FUNCTION_BLOCK LiftModel (* Basic Function Block Type *)
  (* Standard: 61499-2 *)
  (* Version 0.0, 4/20/2019, vshatrov, nxtControl GmbH, Template *)
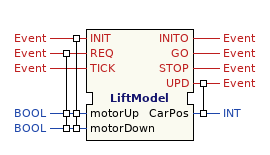
  EVENT_INPUT
    INIT WITH motorUp, motorDown; (* Initialization Request *)
    REQ WITH motorUp, motorDown; (* Normal Execution Request *)
    TICK;
  END_EVENT
  EVENT_OUTPUT
    INITO;
    GO; (* Initialization Confirm *)
    STOP; (* Execution Confirmation *)
    UPD WITH CarPos;
  END_EVENT
  VAR_INPUT
    motorUp : BOOL; (* Input event qualifier *)
    motorDown : BOOL;
  END_VAR
  VAR_OUTPUT
    CarPos : INT; (* Output event qualifier *)
  END_VAR
  VAR
    Position : DINT;
    direction : DINT;
  END_VAR
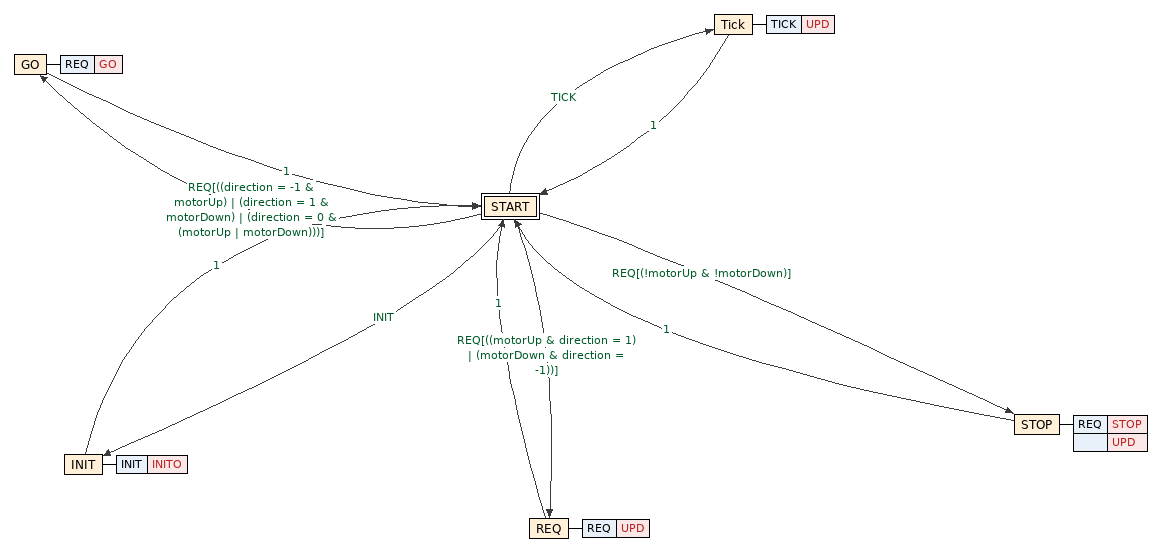
  EC_STATES
    START; (* Initial State *)
    INIT : INIT -> INITO; (* Initialization *)
    REQ : REQ -> UPD; (* Normal execution *)
    Tick : TICK -> UPD;
    GO : REQ -> GO;
    STOP : REQ -> STOP, -> UPD;
  END_STATES
  EC_TRANSITIONS
    START TO INIT := INIT;
    INIT TO START := 1;
    START TO GO := REQ[((direction = -1 & motorUp) | (direction = 1 & motorDown) | (direction = 0 & (motorUp | motorDown)))];
    START TO Tick := TICK;
    Tick TO START := 1;
    START TO STOP := REQ[(!motorUp & !motorDown)];
    GO TO START := 1;
    STOP TO START := 1;
    START TO REQ := REQ[((motorUp & direction = 1) | (motorDown & direction = -1))];
    REQ TO START := 1;
  END_TRANSITIONS
  ALGORITHM INIT IN ST: (* Initialization algorithm *)
;

Position := 1; (*Floor 0*)
direction := 0;
CarPos := Position;
  END_ALGORITHM
  ALGORITHM REQ IN ST: (* Normally executed algorithm *)
IF motorUp THEN
 direction := 1;
ELSIF motorDown THEN
  direction := -1;
ELSE
  direction := 0;
END_IF;
CarPos := Position;
  END_ALGORITHM
  ALGORITHM TICK IN ST:
Position := LIMIT(0, Position + direction, 6);
CarPos := Position;
  END_ALGORITHM
END_FUNCTION_BLOCK
